# EPICS autosave request: soft_iocs/galil_DMC/iocBoot/iocgalil_DMC_E06_08/slit_settings.req
file "2slit_soft_settings.req", P=$(P), SLIT=JJ_D_V:
file "2slit_soft_settings.req", P=$(P), SLIT=JJ_D_H:
